// TwinCAT 3 PLC project DataTypesPLC
// ProgramVersion: 3.1.4024.0
// libraries:
//   Tc2_Standard, * (Beckhoff Automation GmbH)
//   Tc2_System, * (Beckhoff Automation GmbH)
//   Tc3_Module, * (Beckhoff Automation GmbH)
// project tree:
//   / PlcTask.TcTTO
//   POUs/ MAIN.TcPOU
// real-time tasks:
//   TASK PlcTask: cycle T#10ms, priority 20, ADS port 350

CONFIGURATION DataTypesPLC
    RESOURCE PLC ON TwinCAT3
        TASK PlcTask(INTERVAL := T#10ms, PRIORITY := 20);
        PROGRAM MAIN WITH PlcTask : MAIN;
    END_RESOURCE
END_CONFIGURATION

// ---- POUs/MAIN.TcPOU
PROGRAM MAIN
VAR
	IntVAr : INT;
	StrVar : STRING;
	FloatVar : REAL;
	RetunBytesINT : UDINT;
	RetunBytesSTR : UDINT;
	RetunBytesF : UDINT;
	
	nVariable : INT := 20;
	pPointer : POINTER TO INT := ADR(nVariable);
	RetunBytesPtr : UDINT;
	
	Variable : INT := 20;
	rReference : REFERENCE TO INT REF= Variable;
	RetunBytesRef : UDINT;
	aArray : ARRAY [1..5] OF INT := [10, 20, 30, 40, 50];
	nINT : INT;
END_VAR

RetunBytesINT := SIZEOF(IntVAr);
RetunBytesSTR := SIZEOF(StrVar);
RetunBytesF := SIZEOF(FloatVar);

pPointer^ := 30;
RetunBytesPtr := SIZEOF(pPointer);

rReference := 30;
RetunBytesRef := SIZEOF(rReference);

aArray[1] := 42;
nINT := aArray[1] + aArray[4];

END_PROGRAM
